{attribute 'qualified_only'}
VAR_GLOBAL CONSTANT
	INDEX_START 	: INT := 0;	
	MAX_DIMM_LAMPS 	: INT := 14;
	MAX_ONOFF_LAMPS : INT := 14;	
	MAX_LAMPS		: INT := 29;
END_VAR

(* stored: Version 1.1.0.1, ProductVersion 3.1.4024.6
   GVL Param: Id {b9685460-6ce4-4b5a-8e42-d5217ad21500} *)
